% RSLogix 500 project DEMUX.RSS, saved by version 8.30.00.16 %
PROJECT "UNTITLED"    % processor: Bul.1763 MicroLogix 1100 Series B %

PROGRAM FILES
  LAD 2   9 rungs

DATA FILES
  O0 OUTPUT  4 elements
  I1 INPUT  6 elements
  S2 STATUS  66 elements
  B3 BINARY  1 elements
  T4 TIMER  1 elements
  C5 COUNTER  1 elements
  R6 CONTROL  1 elements
  N7 INTEGER  1 elements
  F8 FLOAT  1 elements

LADDER 2
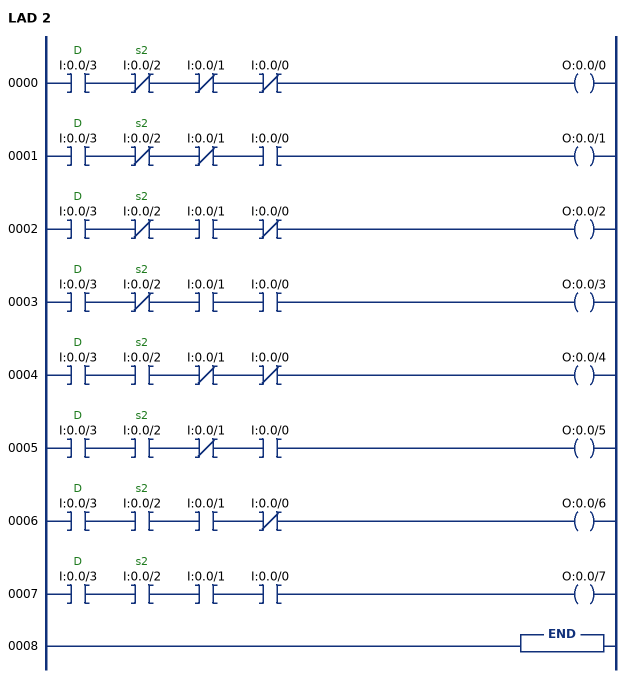
% Rung: 0 %
SOR XIC I:0.0/3 XIO I:0.0/2 XIO I:0.0/1 XIO I:0.0/0 OTE O:0.0/0 EOR
%   I:0.0/3  D %
%   I:0.0/2  "s2" %
%   XIO I:0.0/2  "s2" %
%   XIO I:0.0/1  "s1" %
%   XIO I:0.0/0  "s0" %
% Rung: 1 %
SOR XIC I:0.0/3 XIO I:0.0/2 XIO I:0.0/1 XIC I:0.0/0 OTE O:0.0/1 EOR
%   I:0.0/3  D %
%   I:0.0/2  "s2" %
%   XIO I:0.0/2  "s2" %
%   XIO I:0.0/1  "s1" %
%   XIC I:0.0/0  "s0" %
% Rung: 2 %
SOR XIC I:0.0/3 XIO I:0.0/2 XIC I:0.0/1 XIO I:0.0/0 OTE O:0.0/2 EOR
%   I:0.0/3  D %
%   I:0.0/2  "s2" %
%   XIO I:0.0/2  "s2" %
%   XIC I:0.0/1  "s1" %
%   XIO I:0.0/0  "s0" %
% Rung: 3 %
SOR XIC I:0.0/3 XIO I:0.0/2 XIC I:0.0/1 XIC I:0.0/0 OTE O:0.0/3 EOR
%   I:0.0/3  D %
%   I:0.0/2  "s2" %
%   XIO I:0.0/2  "s2" %
%   XIC I:0.0/1  "s1" %
%   XIC I:0.0/0  "s0" %
% Rung: 4 %
SOR XIC I:0.0/3 XIC I:0.0/2 XIO I:0.0/1 XIO I:0.0/0 OTE O:0.0/4 EOR
%   I:0.0/3  D %
%   I:0.0/2  "s2" %
%   XIO I:0.0/1  "s1" %
%   XIO I:0.0/0  "s0" %
% Rung: 5 %
SOR XIC I:0.0/3 XIC I:0.0/2 XIO I:0.0/1 XIC I:0.0/0 OTE O:0.0/5 EOR
%   I:0.0/3  D %
%   I:0.0/2  "s2" %
%   XIO I:0.0/1  "s1" %
%   XIC I:0.0/0  "s0" %
% Rung: 6 %
SOR XIC I:0.0/3 XIC I:0.0/2 XIC I:0.0/1 XIO I:0.0/0 OTE O:0.0/6 EOR
%   I:0.0/3  D %
%   I:0.0/2  "s2" %
%   XIC I:0.0/1  "s1" %
%   XIO I:0.0/0  "s0" %
% Rung: 7 %
SOR XIC I:0.0/3 XIC I:0.0/2 XIC I:0.0/1 XIC I:0.0/0 OTE O:0.0/7 EOR
%   I:0.0/3  D %
%   I:0.0/2  "s2" %
%   XIC I:0.0/1  "s1" %
%   XIC I:0.0/0  "s0" %
% Rung: 8 %
SOR END EOR
